# EPICS StreamDevice protocol: b17tmagSup/b17tmag.proto
InTerminator = "\r\n";
OutTerminator = "\r";

ReplyTimeout = 2000;

getField {
    out "output";
    in "output:OK:%(\$1FIELD)fT,%f(\$1CURR)A";
}

getHeater {
    out "heater";
    in "heater:OK:[0-3]";
}

# NEED TO FIX
getPersist {
    out "persistent";
    # in "%(\$1FIELD:PERSIST),%f(\$1CURR:PERSIST)";
    in "persistent:OK:%(\$1FIELD:PERSIST)fT,%f(\$1CURR:PERSIST)A";
}

# getPersistMode {
#     out "persistmode";
#     in "persistmode:OK:/^(ON|OFF)$/";
# }
getPersistMode {
    out "persistmode";
    in "persistmode:OK:%s";
}

getReady {
    out "ready";
    in "ready:OK:/^(ON|OFF)$/";
}

getSensA {
    out "sensA";
    in "sensA:OK:[0-9]*\.[0-9]";
}

# NEED TO FIX - FIXED? removed "+" from end of in line for A and B
getSensB {
    out "sensB";
    in "sensB:OK:[0-9]*\.[0-9]";
}

setField {
    out "abort";
    out "setfield:\d";
    in "setfield:\d";
}

setPersistMode {
    out "setpersist %{OFF|ON}";
    in "setpersist:%s";
}
# setPersistMode {
#     out "setpersist %{OFF|ON}";
#     in "setpersist: %{OFF|ON}";
# }

# getTempA {
#     out "sensA";
#     in "sensA:OK:\d";
# }

# getTempB {
#     out "sensB";
#     in "sensB:OK:\d";
# }

getSet1 {
    out "setpoint1";
    in "setpoint1:OK:\f";
}

# NEED TO FIX - fixed incorrect spelling in device file
getSet2 {
    out "setpoint2";
    in "setpoint2:OK:\f";
}

setSet1 {
    out "set1\d";
    in "set1:\d";
}

setSet2 {
    out "set2\d";
    in "set2:\d";
}

# NEED TO FIX
getNeedlePosition {
    out "nv";
    in "nv:OK:\d";
}

getPressure {
    out "pressure";
    in "output:OK:%(\$1NV:PRESSURE:SP:RBV)f,%f(\$1NV:PRESSURE)f";
}

setPressure {
    out "setpressure[0-9]*\.[0-9]+";
    in "setpressure:[0-9]*\.[0-9]+";
}

setNeedlePosition {
    out "setposition[0-9]*\.[0-9]+";
    in "setposition:[0-9]*\.[0-9]+";
}

getAttoAngle {
    out "attoangle";
    in "attoangle:OK:[0-2]?[0-9]{1,2}.[0-9]?{2}|3[0-5][0-9].[0-9]?{2}|360.00)";
}

getHelLevel {
    out "helevel";
    in "helevel:OK:\d";
}

setAttoAngle {
    out "setangle\f";
    in "setangle:\s";
}

# NEED TO FIX - Fixed was not
# connected correctly and moved output to one line return as newline did not work
getMacroStatus {
    out "getstatus";
    in "getstatus:OK:\s";
}
